FUNCTION_BLOCK Test_TExecutionWhenBusy_SetAborted_RaisesNotification EXTENDS T_UnitTestbase
VAR
    Execution                            : T_Execution;
    ExecutionFailed_NotificationHandler  : T_NotificationHandler;
    ExecutionAborted_NotificationHandler : T_NotificationHandler;
END_VAR

METHOD Init
// Setup...
Execution.FB_init(bInitRetains := FALSE,
                  bInCopyCode  := FALSE);

ExecutionFailed_NotificationHandler.FB_init(bInitRetains := FALSE,
                                            bInCopyCode  := FALSE);

ExecutionAborted_NotificationHandler.FB_init(bInitRetains := FALSE,
                                             bInCopyCode  := FALSE);
END_METHOD

{attribute 'analysis' := '-33'} // inhibit unused variable warning
METHOD RunTest
VAR_OUTPUT
    TestCompleted : BOOL;
    TestFailed    : BOOL;
END_VAR
// link handler to common execution events...
GlobalNotifications.Notification_ExecutionFailed
    .ClearNotificationHandlers()
    .AddNotificationHandler(ExecutionFailed_NotificationHandler);

GlobalNotifications.Notification_ExecutionAborted
    .ClearNotificationHandlers()
    .AddNotificationHandler(ExecutionAborted_NotificationHandler);

// Test...
Execution.Start();
Execution.SetBusy();
Execution.SetAborted(); // raises error event

TestFailed S= NOT AssertTrue(Source    := TestName,
                             Condition := ExecutionAborted_NotificationHandler.IsRaised(),
                             Message   := 'ExecutionAborted_NotificationHandler.IsRaised() not true');

TestCompleted := TRUE;
END_METHOD

END_FUNCTION_BLOCK

(* stored: Version 1.1.0.1, ProductVersion 3.1.4024.12
   POU Test_TExecutionWhenBusy_SetAborted_RaisesNotification: Id {686cfdfe-2411-449f-8f4c-b33e4c8bd5de}, SpecialFunc None
   Method Init: Id {e635a7d1-892f-4bcc-80e8-2ae237436d52}
   Method RunTest: Id {36922624-a851-432e-be68-79ecc33aad86} *)
